Staubli VAL3: goTo.pgx

public program goTo(tool x_tTool, mdesc x_mDesc, num x_nMoveType, bool& x_bUnreached[], num x_nIndex)
  local mdesc temp_mdesc
  local num l_nSize
  local point l_pPoint
  local joint l_jJoint
  local frame l_ZoneFrame
  local bool l_bCheck
  local num l_nType
  local num l_nDimension
  local tool l_tTool
  local string l_sMessage
  local num l_nMoveId
begin
  // check for the zone
  if (jEditPoint.nZoneType!=0 and x_nIndex==0) or find(jEditPoint.tData[x_nIndex].tSuper.comment,"@")!=-1
    // take the tool
    // use flange
    l_tTool=flange
    //call tcp:getTool(l_tTool,jEditPoint.nIndexTool)
    // take the three points
    pPoints[0]=jEditPoint.pO
    pPoints[1]=jEditPoint.pX
    pPoints[2]=jEditPoint.pY
    // take the distance
    l_nDimension=jEditPoint.nDimension
    //take the type
    l_nType=jEditPoint.nZoneType
    // check the frame type-2 CIRCLE
    if setFrame(pPoints[0],pPoints[1],pPoints[2],fSetFrame)==0 or l_nType==2
      call checkZone(pPoints,l_tTool,l_nDimension,l_nType,l_bCheck)
      // show the result
      if l_bCheck
        // inside the zone
        call language:message(l_sMessage,225)
        // move TO
        call moveTo(l_tTool,x_mDesc,x_nMoveType,x_bUnreached,x_nIndex,l_nMoveId,false)
      elseIf find(jEditPoint.tData[x_nIndex].tSuper.comment,"@")!=-1
        // link POINT
        // look for the moveType
        call findMove(x_nIndex,l_tTool,x_nMoveType)
        call moveTo(l_tTool,x_mDesc,x_nMoveType,x_bUnreached,x_nIndex,l_nMoveId,false)
      else
        //outside the zone
        call language:message(l_sMessage,226)
      endIf
    elseIf find(jEditPoint.tData[x_nIndex].tSuper.comment,"@")!=-1
      // found a @POINT-JPOINT
      call moveTo(l_tTool,x_mDesc,x_nMoveType,x_bUnreached,x_nIndex,l_nMoveId,false)
    else
      // frame not define
      call language:message(l_sMessage,183)
      call use:timerDialog(l_sMessage,3)
    endIf
  elseIf isInRange(jEditPoint.tData[x_nIndex].jJoint)
    // look for the moveType
    call findMove(x_nIndex,x_tTool,x_nMoveType)
    // execute the movement
    switch x_nMoveType
      case 0
        // JOINT MOVE
        // go to the select Joint
        movej(jEditPoint.tData[x_nIndex].jJoint,x_tTool,x_mDesc)
      break
      case 1
        // LINEAR MOVE
        movel(jointToPoint(x_tTool,world,jEditPoint.tData[x_nIndex].jJoint),x_tTool,x_mDesc)
      break
      default
      break
    endSwitch
  else
    x_bUnreached=true
  endIf
  // save the actual index
  nIndex=x_nIndex
end
